FUNCTION_BLOCK FB_PLUS
VAR_INPUT
	inValue01:REAL;
	inValue02:REAL;
END_VAR
VAR_OUTPUT
	outSum:REAL;
END_VAR
VAR
	Val01_Local:REAL;
	Val02_Local:REAL;
	Sum_Local:REAL;
END_VAR

Val01_Local:=inValue01;
Val02_Local:=inValue02;

Sum_Local:=Val01_Local+Val02_Local;

outSum:=Sum_Local;

END_FUNCTION_BLOCK

(* stored: Version 1.1.0.1, ProductVersion 3.1.4024.4
   POU FB_PLUS: Id {884e3b13-609c-4f51-9059-3c29986c0898}, SpecialFunc None *)
